{attribute 'qualified_only'}
VAR_GLOBAL
	DoTest : BOOL;
END_VAR

(* stored: Version 1.1.0.1, ProductVersion 3.1.4024.9
   GVL Inputs: Id {b040d1d9-8e59-4fa8-97ed-e7fbf86322ce} *)
